// TIA Portal V18 export
FUNCTION_BLOCK "axis_manager"   // FB25, FBD
{ S7_Optimized_Access := 'TRUE' }
VERSION : 0.1
// stored: AutoNumber true, IsIECCheckEnabled false, IsRetainMemResEnabled false, MemoryReserve 100, SetENOAutomatically false, UDAEnableTagReadback false
   VAR_INPUT
      allowed : Bool;
      targetUnison : Real;
      targetHome : Real;
      targetStep : Real;
      bSoftStop : Bool;
      bHome : Bool;
      hbStepPlus : Bool;
      hbStepMinus : Bool;
      bFwd : Bool;
      bRev : Bool;
      Params : "typeMotPara";
      ExecUni : Bool;
      theseAreDoors : Bool;
      xOverrideLOCAL : Bool;
      POS : Real;
   END_VAR
   VAR_OUTPUT
      team_unison : Bool;
      team_free : Bool;
      team_override : Bool;
      Desk_slowly : Bool;
      yaSpeedManual : Real;
      yaSpeedAuto : Real;
      m_auto : Bool;
      m_man : Bool;
      au_execute : Bool;
      aut_target : Real;
      OVERRIDE : Bool;
      ExecutingManuverFreeMode : Bool;
   END_VAR
   VAR
      st_Fwd : Bool;
      st_Rev : Bool;
      st_speed_slow_or_fast_negative : Real;
      aman_sel_target_Instance { S7_SetPoint := 'True'} : "aman_sel_target";
   END_VAR
   VAR_TEMP
      st_speedManual_slow_or_fast : Real;
      SpeedBlind : Real;
      stSpeedManualSlow : Real;
      Speed_autoSlow : Real;
   END_VAR
BEGIN

REGION Network 1
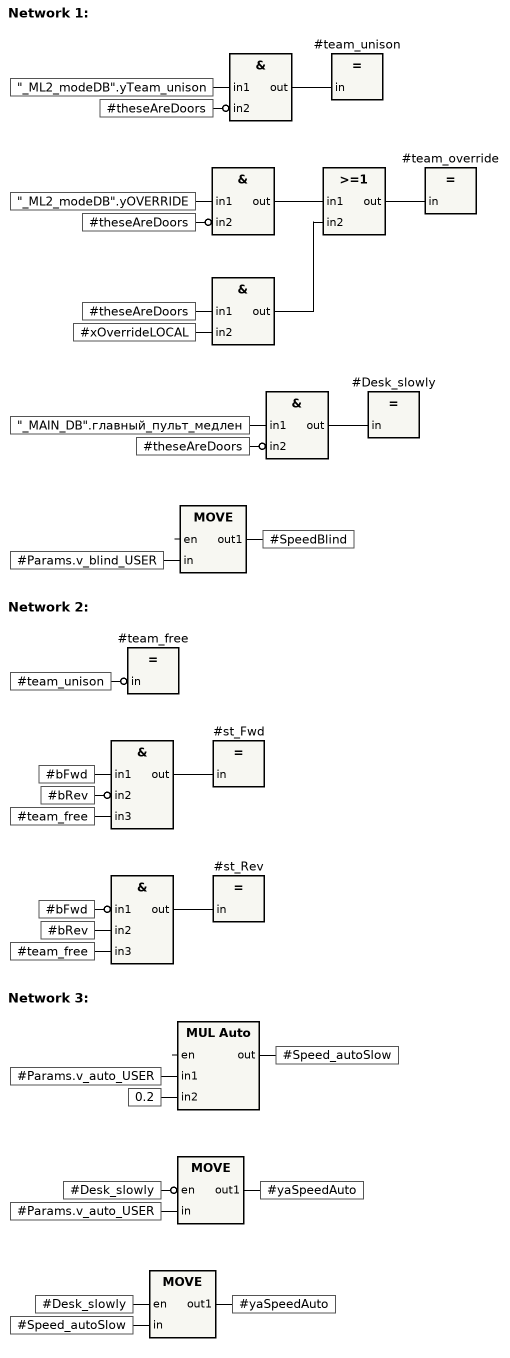
   #team_unison := "_ML2_modeDB".yTeam_unison AND NOT #theseAreDoors;
   #team_override := ("_ML2_modeDB".yOVERRIDE AND NOT #theseAreDoors) OR (#theseAreDoors AND #xOverrideLOCAL);
   #Desk_slowly := "_MAIN_DB".главный_пульт_медлен AND NOT #theseAreDoors;
   #SpeedBlind := #Params.v_blind_USER;
END_REGION

REGION Network 2
   #team_free := NOT #team_unison;
   #st_Fwd := #bFwd AND NOT #bRev AND #team_free;
   #st_Rev := NOT #bFwd AND #bRev AND #team_free;
END_REGION

REGION Network 3
   #Speed_autoSlow := #Params.v_auto_USER * 0.2;
   IF NOT #Desk_slowly THEN #yaSpeedAuto := #Params.v_auto_USER; END_IF;
   IF #Desk_slowly THEN #yaSpeedAuto := #Speed_autoSlow; END_IF;
END_REGION

REGION Network 4
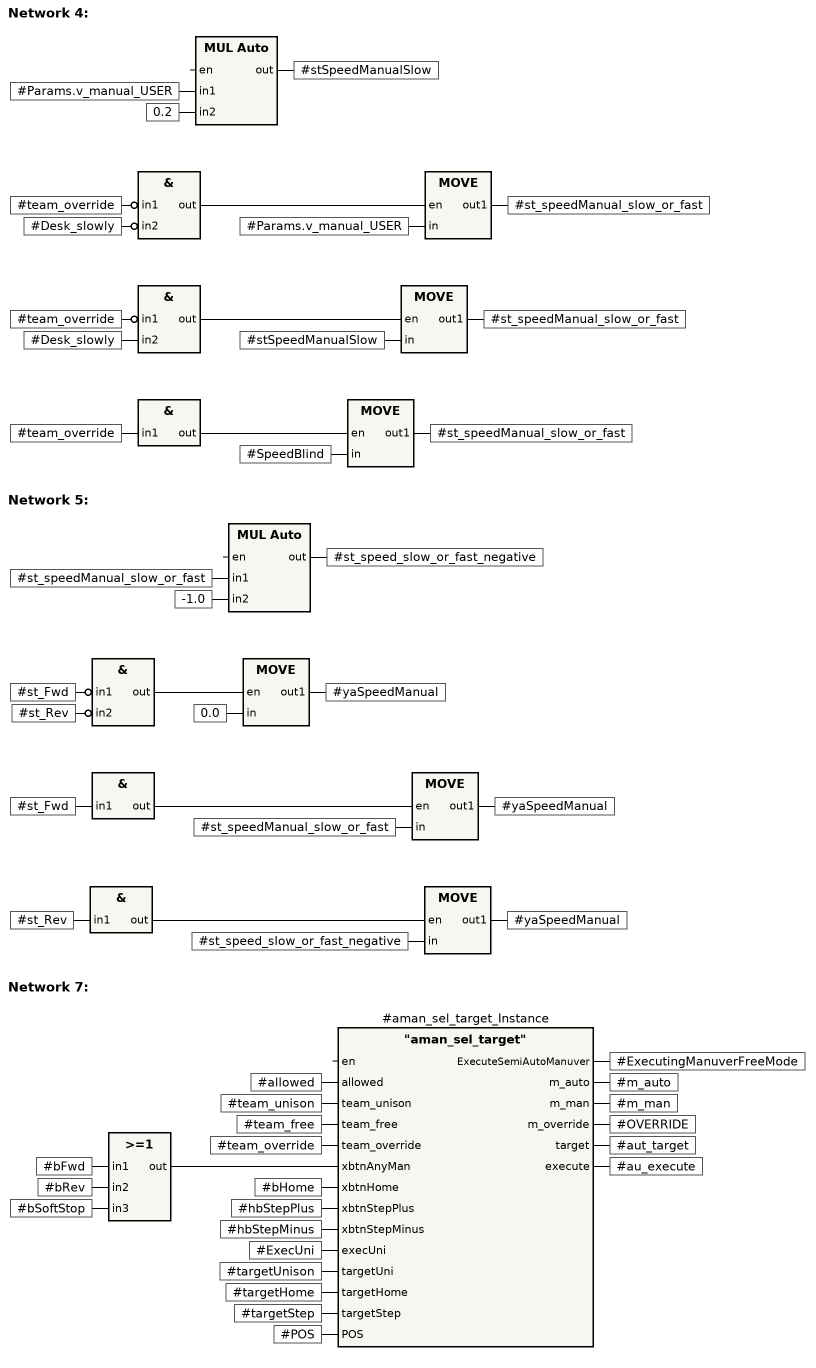
   #stSpeedManualSlow := #Params.v_manual_USER * 0.2;
   IF NOT #team_override AND NOT #Desk_slowly THEN
       #st_speedManual_slow_or_fast := #Params.v_manual_USER;
   END_IF;
   IF NOT #team_override AND #Desk_slowly THEN #st_speedManual_slow_or_fast := #stSpeedManualSlow; END_IF;
   IF #team_override THEN #st_speedManual_slow_or_fast := #SpeedBlind; END_IF;
END_REGION

REGION Network 5
   #st_speed_slow_or_fast_negative := #st_speedManual_slow_or_fast * (-1.0);
   IF NOT #st_Fwd AND NOT #st_Rev THEN #yaSpeedManual := 0.0; END_IF;
   IF #st_Fwd THEN #yaSpeedManual := #st_speedManual_slow_or_fast; END_IF;
   IF #st_Rev THEN #yaSpeedManual := #st_speed_slow_or_fast_negative; END_IF;
END_REGION

REGION Network 7
   #aman_sel_target_Instance(allowed := #allowed,   // "aman_sel_target"
                           team_unison := #team_unison,
                           team_free := #team_free,
                           team_override := #team_override,
                           xbtnAnyMan := #bFwd OR #bRev OR #bSoftStop,
                           xbtnHome := #bHome,
                           xbtnStepPlus := #hbStepPlus,
                           xbtnStepMinus := #hbStepMinus,
                           execUni := #ExecUni,
                           targetUni := #targetUnison,
                           targetHome := #targetHome,
                           targetStep := #targetStep,
                           POS := #POS,
                           ExecuteSemiAutoManuver => #ExecutingManuverFreeMode,
                           m_auto => #m_auto,
                           m_man => #m_man,
                           m_override => #OVERRIDE,
                           target => #aut_target,
                           execute => #au_execute);
END_REGION
END_FUNCTION_BLOCK
